% RSLogix 500 project Digital-Control-Logic.RSS, saved by version 8.30.00.16 %
PROJECT "MICRO"    % processor: Bul.1763 MicroLogix 1100 Series B %

PROGRAM FILES
  LAD 2 "MAIN"  3 rungs
  LAD 3 "I/O"  5 rungs  % InputOutput %
  LAD 4 "LOGIC"  6 rungs  % PROGRAM LOGIC %

DATA FILES
  O0 OUTPUT  4 elements
  I1 INPUT  6 elements
  S2 STATUS  66 elements
  B3 BINARY  4 elements
  T4 TIMER  1 elements
  C5 COUNTER  1 elements
  R6 CONTROL  1 elements
  N7 INTEGER  1 elements
  F8 FLOAT  1 elements

LADDER 2 "MAIN"
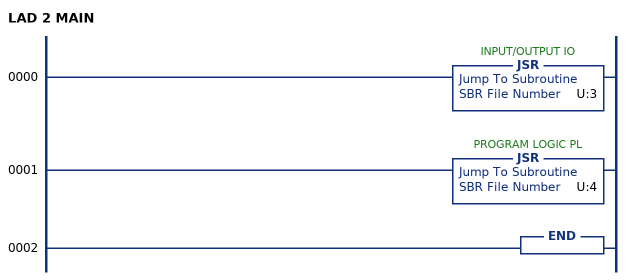
% Rung: 0 %
SOR JSR U:3 EOR
%   U:3  IO  "INPUT/OUTPUT" %
% Rung: 1 %
SOR JSR U:4 EOR
%   U:4  PL  "PROGRAM LOGIC" %
% Rung: 2 %
SOR END EOR

LADDER 3 "I/O"    % InputOutput %
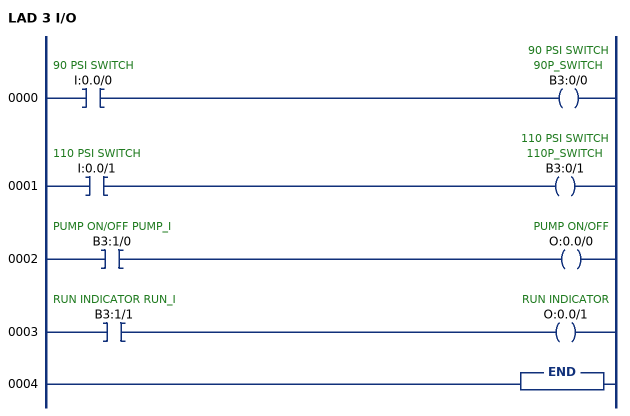
% Rung: 0 %
SOR XIC I:0.0/0 OTE B3:0/0 EOR
%   I:0.0/0  "90 PSI SWITCH" %
%   B3:0/0  90P_SWITCH  "90 PSI SWITCH" %
% Rung: 1 %
SOR XIC I:0.0/1 OTE B3:0/1 EOR
%   I:0.0/1  "110 PSI SWITCH" %
%   B3:0/1  110P_SWITCH  "110 PSI SWITCH" %
% Rung: 2 %
SOR XIC B3:1/0 OTE O:0.0/0 EOR
%   B3:1/0  PUMP_I  "PUMP ON/OFF" %
%   O:0.0/0  "PUMP ON/OFF" %
% Rung: 3 %
SOR XIC B3:1/1 OTE O:0.0/1 EOR
%   B3:1/1  RUN_I  "RUN INDICATOR" %
%   O:0.0/1  "RUN INDICATOR" %
% Rung: 4 %
SOR END EOR

LADDER 4 "LOGIC"    % PROGRAM LOGIC %
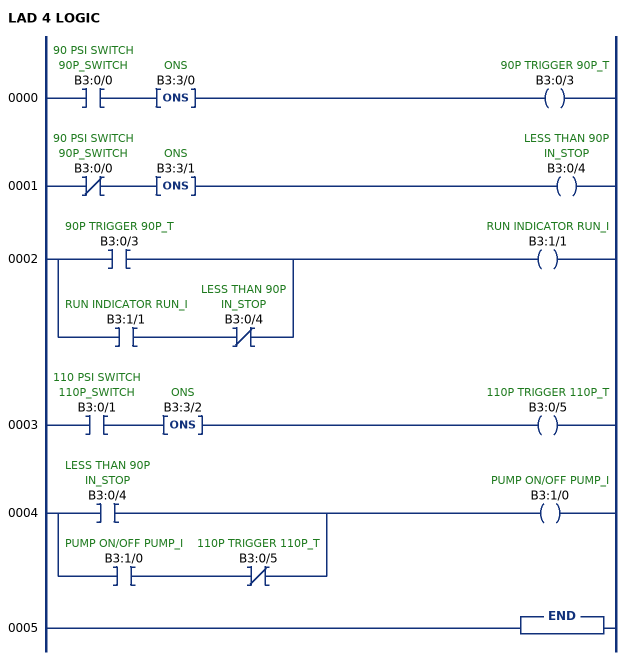
% Rung: 0 %  % edit flag set %
SOR XIC B3:0/0 ONS B3:3/0 OTE B3:0/3 EOR
%   B3:0/0  90P_SWITCH  "90 PSI SWITCH" %
%   B3:3/0  "ONS" %
%   B3:0/3  90P_T  "90P TRIGGER" %
% Rung: 1 %  % edit flag set %
SOR XIO B3:0/0 ONS B3:3/1 OTE B3:0/4 EOR
%   B3:0/0  90P_SWITCH  "90 PSI SWITCH" %
%   B3:3/1  "ONS" %
%   B3:0/4  IN_STOP  "LESS THAN 90P" %
% Rung: 2 %
SOR BST XIC B3:0/3 NXB XIC B3:1/1 XIO B3:0/4 BND OTE B3:1/1 EOR
%   B3:0/3  90P_T  "90P TRIGGER" %
%   B3:1/1  RUN_I  "RUN INDICATOR" %
%   B3:0/4  IN_STOP  "LESS THAN 90P" %
% Rung: 3 %  % edit flag set %
SOR XIC B3:0/1 ONS B3:3/2 OTE B3:0/5 EOR
%   B3:0/1  110P_SWITCH  "110 PSI SWITCH" %
%   B3:3/2  "ONS" %
%   B3:0/5  110P_T  "110P TRIGGER" %
% Rung: 4 %
SOR BST XIC B3:0/4 NXB XIC B3:1/0 XIO B3:0/5 BND OTE B3:1/0 EOR
%   B3:0/4  IN_STOP  "LESS THAN 90P" %
%   B3:1/0  PUMP_I  "PUMP ON/OFF" %
%   B3:0/5  110P_T  "110P TRIGGER" %
% Rung: 5 %
SOR END EOR

OTHER DOCUMENTED ADDRESSES
  B3:2/0  "ONS"
  B3:2/1  "ONS"
  B3:2/2  "ONS"
  B3:2/3  "ONS"
  B3:3/3  "ONS"

DATA TABLE (non-zero values as saved)
DATA B3
% B3:0 % 0X0000 0X0001 0X0001 0X0008
